// TwinCAT 3 PLC project PLC1
// ProgramVersion: 3.1.4024.0
// libraries:
//   Tc2_DataExchange, * (Beckhoff Automation GmbH)
//   Tc2_Standard, * (Beckhoff Automation GmbH)
//   Tc2_System, * (Beckhoff Automation GmbH)
//   Tc3_Module, * (Beckhoff Automation GmbH)
// project tree:
//   GVLs/ GVL_Tank.TcGVL, GVL_Tank_Previous.TcGVL
//   / PlcTask.TcTTO
//   POUs/ FB_TankController.TcPOU, FB_UpdateHandler.TcPOU, MAIN.TcPOU
// real-time tasks:
//   TASK PlcTask: cycle T#10ms, priority 20, ADS port 350
//   TASK PlcTask1: cycle T#10ms, priority 21, ADS port 351

CONFIGURATION PLC1
    RESOURCE PLC ON TwinCAT3
        TASK PlcTask(INTERVAL := T#10ms, PRIORITY := 20);
        PROGRAM MAIN WITH PlcTask : MAIN;
    END_RESOURCE
END_CONFIGURATION

// ---- GVLs/GVL_Tank.TcGVL
{attribute 'qualified_only'}
{attribute 'TcAdsSymEntry'}
VAR_GLOBAL
    nTankLevel      : INT := 0;       // 0-100 percent
    bPumpOn         : BOOL := FALSE;
    bValveOpen      : BOOL := FALSE;
    bOverflow       : BOOL := FALSE;
    bUnderflow      : BOOL := FALSE;
    sStatusMsg      : STRING := 'System Ready';
    bResetAlarm     : BOOL := FALSE;  // PLC2 writes this to reset
END_VAR

// ---- GVLs/GVL_Tank_Previous.TcGVL
{attribute 'qualified_only'}
{attribute 'TcAdsSymEntry'}
VAR_GLOBAL
    nTankLevel_prev      : INT := 0;       // 0-100 percent
    bPumpOn_prev         : BOOL := FALSE;
    bValveOpen_prev      : BOOL := FALSE;
    bOverflow_prev       : BOOL := FALSE;
    bUnderflow_prev      : BOOL := FALSE;
    sStatusMsg_prev      : STRING := 'System Ready';
    bResetAlarm_prev     : BOOL := FALSE;  // PLC2 writes this to reset
END_VAR

// ---- POUs/MAIN.TcPOU
PROGRAM MAIN
VAR
	fbTank : FB_TankController;
	fbHandle : FB_UpdateHandler;
END_VAR

fbTank();
fbHandle();

END_PROGRAM

// ---- POUs/FB_TankController.TcPOU
FUNCTION_BLOCK FB_TankController
VAR
    fbFillTimer     : TON;
    fbDrainTimer    : TON;
    nSimLevel       : INT := 0;
END_VAR



// ── Simulate tank filling when pump is ON ────────────────────────────
fbFillTimer(IN := GVL_Tank.bPumpOn, PT := T#1S);
IF fbFillTimer.Q THEN
    fbFillTimer(IN := FALSE);
    IF nSimLevel < 100 THEN
        nSimLevel := nSimLevel + 5;
    END_IF
END_IF

// ── Simulate tank draining when valve is OPEN ────────────────────────
fbDrainTimer(IN := GVL_Tank.bValveOpen, PT := T#1S);
IF fbDrainTimer.Q THEN
    fbDrainTimer(IN := FALSE);
    IF nSimLevel > 0 THEN
        nSimLevel := nSimLevel - 3;
    END_IF
END_IF

// ── Update level ─────────────────────────────────────────────────────
GVL_Tank.nTankLevel := nSimLevel;

// ── Check overflow ───────────────────────────────────────────────────
IF GVL_Tank.nTankLevel >= 90 THEN
    GVL_Tank.bOverflow   := TRUE;
    GVL_Tank.bPumpOn     := FALSE;   // auto stop pump
    GVL_Tank.sStatusMsg  := 'OVERFLOW WARNING - Pump Stopped';

ELSIF GVL_Tank.nTankLevel <= 10 THEN
    GVL_Tank.bUnderflow  := TRUE;
    GVL_Tank.bValveOpen  := FALSE;   // auto close valve
    GVL_Tank.sStatusMsg  := 'UNDERFLOW WARNING - Valve Closed';

ELSE
    GVL_Tank.bOverflow   := FALSE;
    GVL_Tank.bUnderflow  := FALSE;
    GVL_Tank.sStatusMsg  := 'Running Normal';
END_IF



// ── Reset from PLC2 acknowledgement ──────────────────────────────────
IF GVL_Tank.bResetAlarm THEN
    GVL_Tank.bOverflow      := FALSE;
    GVL_Tank.bUnderflow     := FALSE;
    GVL_Tank.sStatusMsg     := 'Alarm Reset by Operator';
    GVL_Tank.bResetAlarm    := FALSE;
END_IF

END_FUNCTION_BLOCK

// ---- POUs/FB_UpdateHandler.TcPOU
FUNCTION_BLOCK FB_UpdateHandler
VAR
	fbWrite1     :  FB_WriteAdsSymByName;
	bEnable     : BOOL;
	sSymbol     : STRING := 'GVL_Alarm.bOverflow';
	eComMode    :  E_AdsComMode := eAdsComModeFastCom;
	bBusy       : BOOL;
    bError      : BOOL;
    nErrId      : UDINT;
	bExecute: BOOL;
	fbTimer : TON := (PT := T#100MS); // Adjust the speed here
	bTriggerWrite: BOOL;
END_VAR


// 1. Detect Change (Edge Detection)
IF GVL_Tank.bOverflow <> GVL_Tank_Previous.bOverflow_prev AND NOT fbWrite1.bBusy THEN
    bTriggerWrite := TRUE;
    // Update previous value only when we start the write
    GVL_Tank_Previous.bOverflow_prev := GVL_Tank.bOverflow;
END_IF

// 2. Call the Function Block
fbWrite1(
    bWrite   := bTriggerWrite, 
    sNetId   := '', 
    nPort    := 851, // Check if target is 851 or 852
    sVarName := sSymbol, 
    nSrcAddr := ADR(GVL_Tank.bOverflow), 
    nLen     := SIZEOF(GVL_Tank.bOverflow), 
    tTimeout := T#5S
);

// 3. Reset Trigger when finished
//IF NOT fbWrite1.bBusy THEN
  //  bTriggerWrite := FALSE;
//END_IF

METHOD M_UpdateValueByADS : BOOL
VAR_INPUT
END_VAR
END_METHOD

END_FUNCTION_BLOCK
